// TIA Portal V20 export
TYPE "typeSafetyDriveStatus"
// Safety status of drive
// stored: Access Published, IsFailsafeCompliant true, Namespace Safety
   STRUCT
      drive1 { S7_SetPoint := 'True'} : "Safety.typeSafetyDrive";
      drive2 { ExternalWritable := 'False'} : "Safety.typeSafetyDrive";
      drive3 { ExternalWritable := 'False'} : "Safety.typeSafetyDrive";
      drive4 { ExternalWritable := 'False'} : "Safety.typeSafetyDrive";
      drive5 : "Safety.typeSafetyDrive";
      drive6 { ExternalWritable := 'False'} : "Safety.typeSafetyDrive";
      drive7 : "Safety.typeSafetyDrive";
      drive8 : "Safety.typeSafetyDrive";
      drive9 : "Safety.typeSafetyDrive";
      drive10 : "Safety.typeSafetyDrive";
      drive11 : "Safety.typeSafetyDrive";
      drive12 : "Safety.typeSafetyDrive";
      drive13 : "Safety.typeSafetyDrive";
      drive14 : "Safety.typeSafetyDrive";
      drive15 : "Safety.typeSafetyDrive";
      drive16 : "Safety.typeSafetyDrive";
      drive17 : "Safety.typeSafetyDrive";
      drive18 : "Safety.typeSafetyDrive";
      drive19 : "Safety.typeSafetyDrive";
      drive20 : "Safety.typeSafetyDrive";
      drive21 : "Safety.typeSafetyDrive";
      drive22 : "Safety.typeSafetyDrive";
      drive23 : "Safety.typeSafetyDrive";
      drive24 : "Safety.typeSafetyDrive";
      drive25 : "Safety.typeSafetyDrive";
      drive26 : "Safety.typeSafetyDrive";
      drive27 : "Safety.typeSafetyDrive";
      drive28 : "Safety.typeSafetyDrive";
      drive29 : "Safety.typeSafetyDrive";
      drive30 : "Safety.typeSafetyDrive";
      drive31 : "Safety.typeSafetyDrive";
      drive32 : "Safety.typeSafetyDrive";
      drive33 : "Safety.typeSafetyDrive";
      drive34 : "Safety.typeSafetyDrive";
      drive35 : "Safety.typeSafetyDrive";
      drive36 : "Safety.typeSafetyDrive";
      drive37 : "Safety.typeSafetyDrive";
      drive38 : "Safety.typeSafetyDrive";
      drive39 : "Safety.typeSafetyDrive";
      drive40 : "Safety.typeSafetyDrive";
      drive41 : "Safety.typeSafetyDrive";
   END_STRUCT;
END_TYPE
